FUNCTION_BLOCK ValveDynamics
VAR_INPUT
END_VAR
VAR_OUTPUT
END_VAR
VAR
END_VAR

END_FUNCTION_BLOCK

(* stored: Version 1.1.0.1, ProductVersion 3.1.4024.9
   POU ValveDynamics: Id {bdd402cd-9955-422d-9429-c814b00ee090}, SpecialFunc None *)
